TYPE ST_AutoPullOutConveyorCommand EXTENDS ST_CommandBasic :
STRUCT
END_STRUCT
END_TYPE

(* stored: Version 1.1.0.1, ProductVersion 3.1.4024.13
   DUT ST_AutoPullOutConveyorCommand: Id {05a04515-190b-4e4c-acb4-d5c7893a6e01} *)
